// TIA Portal project "Project1" (V15)

(* hardware
DEVICE "S7-1200 station_2"  S7-1200 Station
   slot 0: "Rack_0"  S7-1200 Rack  Rack  V1.0
   slot 1: "PLC_2"  CPU 1214C DC/DC/DC  6ES7 214-1AG40-0XB0  V4.2
DEVICE "PC-System_1"  SIMATIC PC station
   slot 0: "SIMATIC PC station"  Rail  SIMATIC PC-Station  V1.0
      slot 125: "Stationmanager"  Station_Manager  V6.0.4
   slot 1: "HMI_RT_1"  WinCC RT Advanced  6AV2 104-0xxxx-xxxx  15.0.0.0
      slot 33792: "Host interface"  Host interface
   slot 2: "IE general_1"  IE General  IE_CP  V8.2.0
*)

// ===== PLC "PLC_2"  CPU 1214C DC/DC/DC =====

VAR_GLOBAL   // PLC tag table "Default tag table"
   "OFF" AT %I0.1 : Bool;
   "Light" AT %Q0.0 : Bool;
   "ON" AT %I0.0 : Bool;
END_VAR

ORGANIZATION_BLOCK "Main"   // OB1, LAD, ProgramCycle
TITLE = "Main Program Sweep (Cycle)"
{ S7_Optimized_Access := 'TRUE' }
VERSION : 0.1
   VAR_INPUT
      Initial_Call : Bool;   // Initial call of this OB
      Remanence : Bool;   // =True, if remanent data are available
   END_VAR
BEGIN

REGION Network 1
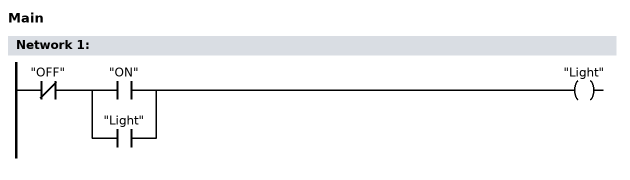
   RUNG wire#powerrail
      I_Contact( "OFF" )
      wire#w1
      Contact( "ON" )
      wire#w2
      Coil( "Light" )
   END_RUNG
   RUNG wire#w1
      Contact( "Light" )
   END_RUNG wire#w2
   // the same network as SCL:
   "Light" := NOT "OFF" AND ("ON" OR "Light");
END_REGION
END_ORGANIZATION_BLOCK

(* ===== HMI "HMI_RT_1" =====
system functions are stored by id; their names below are inferred from use
connection "HMI_Connection_1": ETHERNET, S7_1200_OMS

HMI tags "Default tag table"
   "ON" : Bool = PLC ON AT %I0.0, 1 s
   "OFF" : Bool = PLC OFF AT %I0.1, 1 s
   "Light" : Bool = PLC Light AT %Q0.0, 1 s

screen "Manual" 1024x768
   TextField "Text field_1" at 358,26 size 262x46; Text 'On/Off switch'
   Button "Button_1" at 754,646 size 250x92; TextOff 'Go to Set Up'; TextOn 'Manual'
      on Click: ActivateScreen("Set up", 0)
   Button "Button_2" at 438,646 size 250x92; TextOn 'Manual'; TextOff 'Go to Start'
      on Click: ActivateScreen("Start", 0)

screen "Set up" 1024x768
   TextField "Text field_1" at 358,26 size 262x46; Text 'On/Off switch'
   Button "Button_1" at 754,646 size 250x92; TextOn 'Manual'; TextOff 'Go to Start'
      on Click: ActivateScreen("Start", 0)
   Button "Button_2" at 438,646 size 250x92; TextOn 'Manual'; TextOff 'Go to Manual'
      on Click: ActivateScreen("Manual", 0)

screen "Start" 1024x768
   TextField "Text field_1" at 317,42 size 382x46; Text 'Manual Screen'
   Button "Button_1" at 754,646 size 250x92; TextOn 'Manual'; TextOff 'Go to Set up'
      on Click: ActivateScreen("Set up", 0)
   Button "Button_2" at 438,646 size 250x92; TextOn 'Manual'; TextOff 'Go to Manual'
      on Click: ActivateScreen("Manual", 0)
   Button "Button_3" at 964,6 size 52x46; TextOff 'x'
      on Click: StopRuntime(0)
   Button "Button_4" at 192,188 size 166x118; TextOff 'ON'
      on Press: SetBit("ON")
      on Release: ResetBit("ON")
   Button "Button_5" at 654,182 size 166x118; TextOff 'OFF'
      on Release: ResetBit("OFF")
      on Press: SetBit("OFF")
   Circle "Circle_1" at 462,418 size 84x84
      Appearance <- "Light"
   TextField "Text field_2" at 458,363 size 81x40; Text 'Light'
*)